PROGRAM MAIN
VAR
END_VAR

END_PROGRAM

(* stored: Version 1.1.0.1
   POU MAIN: Id {c1e0513e-f320-4dc5-84ac-ba3d13e16b39} *)
